// SIMATIC S7-200 project (STEP 7-Micro/WIN), CPU 222 REL 02.01

SYMBOL_TABLE 用户定义1
过程值              VD0
设定值              VD4
增益               VD8
采样时间             VD12
积分时间             VD16
微分时间             VD20
PID输出            VD24
积分前项             VD28
过程值前值            VD32
END_SYMBOL_TABLE

ORGANIZATION_BLOCK 主程序:OB1
TITLE=程序注释
BEGIN
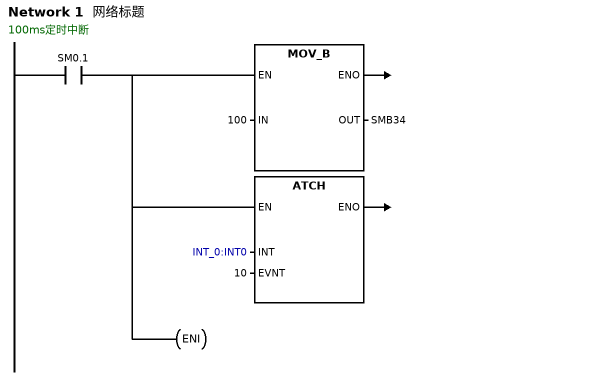
Network 1 // 网络标题
// 100ms定时中断
LD     SM0.1
MOVB   100, SMB34
ATCH   INT_0:INT0, 10
ENI
END_ORGANIZATION_BLOCK

SUBROUTINE_BLOCK PID调用:SBR0
TITLE=子程序注释
VAR_INPUT
过程值:REAL;	// LD0 
设定值:REAL;	// LD4 
增益:REAL;	// LD8 
采样时间:REAL;	// LD12 
积分时间:REAL;	// LD16 
微分时间:REAL;	// LD20 
END_VAR
VAR_IN_OUT
输出值:REAL;	// LD24 
积分前项:REAL;	// LD28 
过程值前值:REAL;	// LD32 
END_VAR
VAR
比例项:REAL;	// LD36 
积分项:REAL;	// LD40 
微分项:REAL;	// LD44 
END_VAR
BEGIN
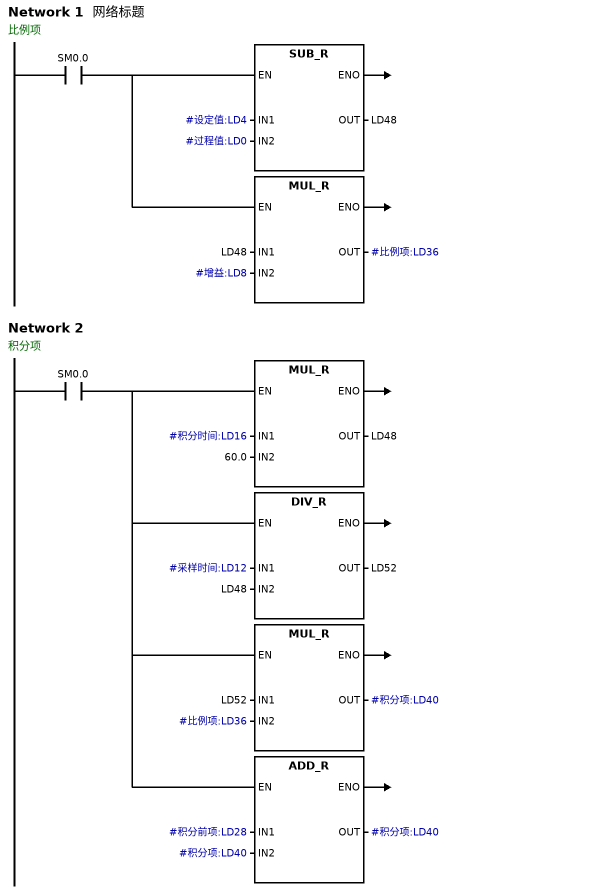
Network 1 // 网络标题
// 比例项
LD     SM0.0
MOVR   #设定值:LD4, LD48
-R     #过程值:LD0, LD48
MOVR   LD48, #比例项:LD36
*R     #增益:LD8, #比例项:LD36
Network 2
// 积分项
LD     SM0.0
MOVR   #积分时间:LD16, LD48
*R     60.0, LD48
MOVR   #采样时间:LD12, LD52
/R     LD48, LD52
MOVR   LD52, #积分项:LD40
*R     #比例项:LD36, #积分项:LD40
+R     #积分前项:LD28, #积分项:LD40
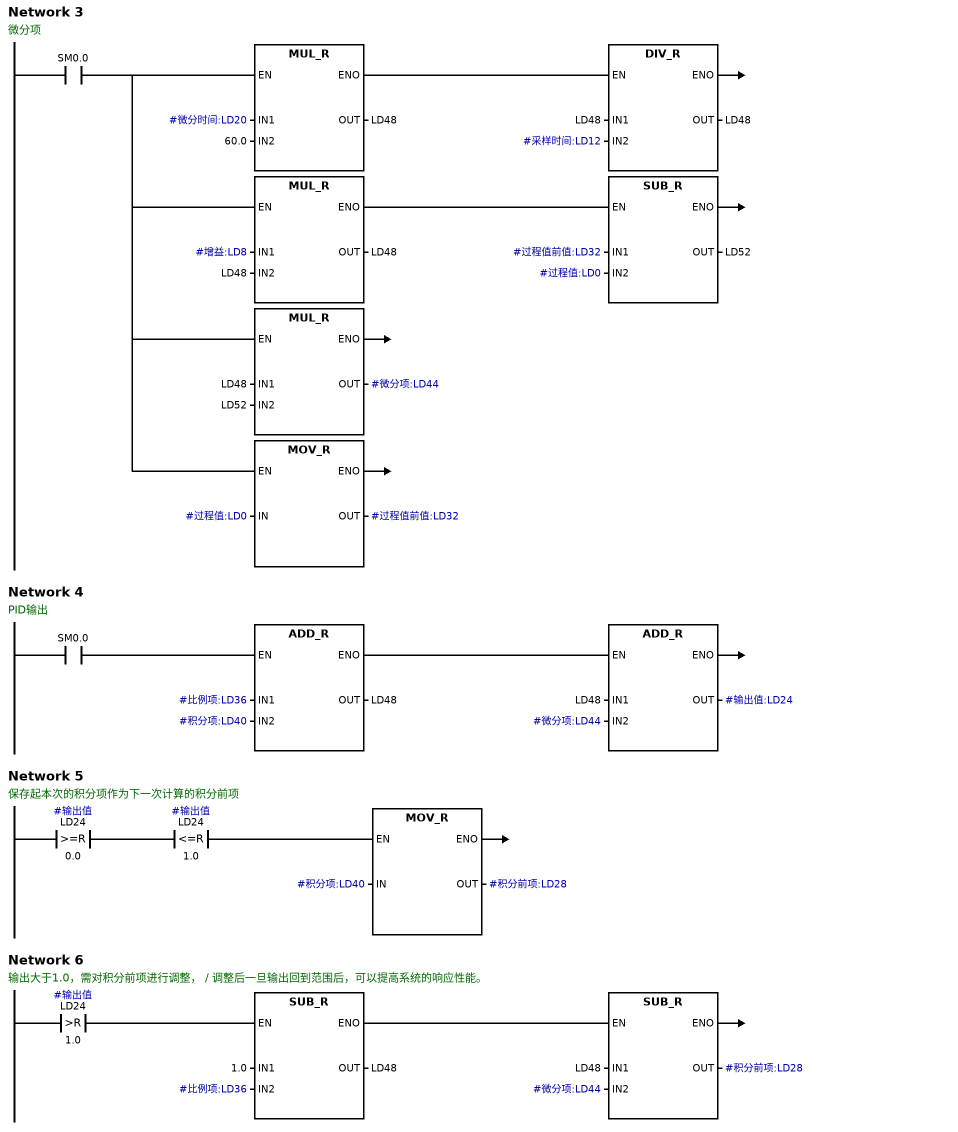
Network 3
// 微分项
LD     SM0.0
LPS
MOVR   #微分时间:LD20, LD48
AENO
*R     60.0, LD48
AENO
/R     #采样时间:LD12, LD48
LRD
*R     #增益:LD8, LD48
AENO
MOVR   #过程值前值:LD32, LD52
-R     #过程值:LD0, LD52
LRD
MOVR   LD48, #微分项:LD44
*R     LD52, #微分项:LD44
LPP
MOVR   #过程值:LD0, #过程值前值:LD32
Network 4
// PID输出
LD     SM0.0
MOVR   #比例项:LD36, LD48
AENO
+R     #积分项:LD40, LD48
AENO
MOVR   LD48, #输出值:LD24
+R     #微分项:LD44, #输出值:LD24
Network 5
// 保存起本次的积分项作为下一次计算的积分前项
LDR>=  #输出值:LD24, 0.0
AR<=   #输出值:LD24, 1.0
MOVR   #积分项:LD40, #积分前项:LD28
Network 6
// 输出大于1.0，需对积分前项进行调整，
// 调整后一旦输出回到范围后，可以提高系统的响应性能。
LDR>   #输出值:LD24, 1.0
MOVR   1.0, LD48
AENO
-R     #比例项:LD36, LD48
AENO
MOVR   LD48, #积分前项:LD28
-R     #微分项:LD44, #积分前项:LD28
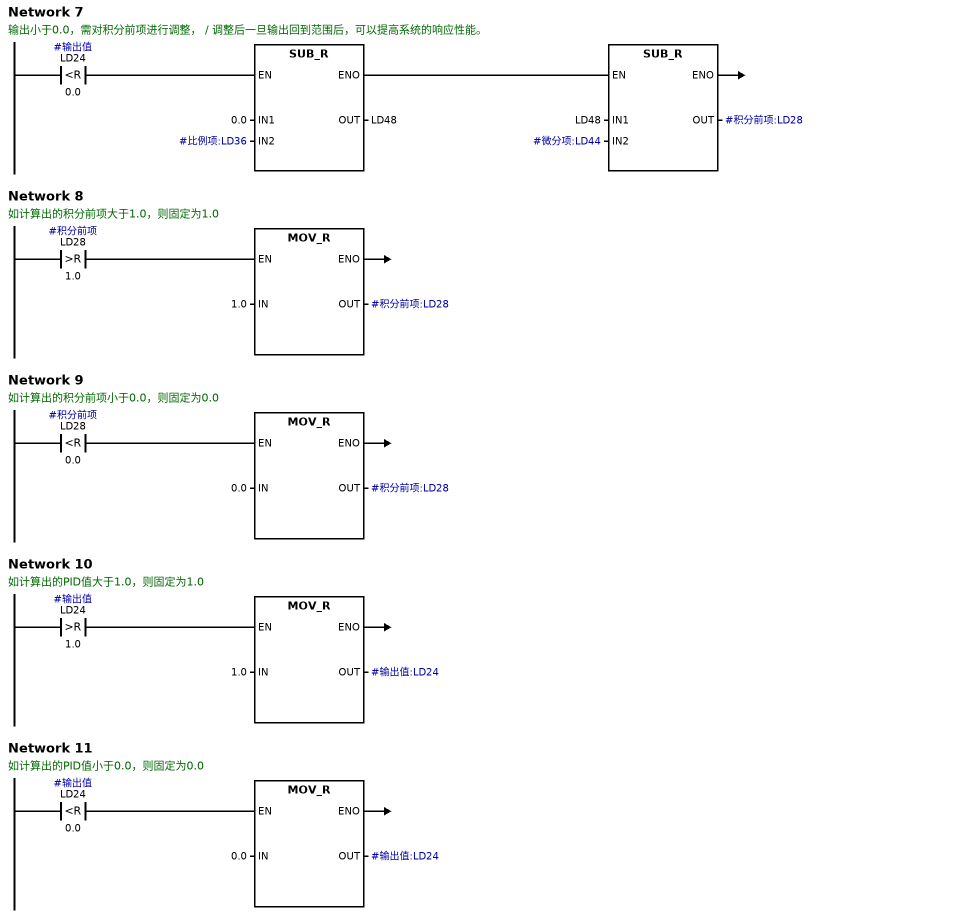
Network 7
// 输出小于0.0，需对积分前项进行调整，
// 调整后一旦输出回到范围后，可以提高系统的响应性能。
LDR<   #输出值:LD24, 0.0
MOVR   0.0, LD48
AENO
-R     #比例项:LD36, LD48
AENO
MOVR   LD48, #积分前项:LD28
-R     #微分项:LD44, #积分前项:LD28
Network 8
// 如计算出的积分前项大于1.0，则固定为1.0
LDR>   #积分前项:LD28, 1.0
MOVR   1.0, #积分前项:LD28
Network 9
// 如计算出的积分前项小于0.0，则固定为0.0
LDR<   #积分前项:LD28, 0.0
MOVR   0.0, #积分前项:LD28
Network 10
// 如计算出的PID值大于1.0，则固定为1.0
LDR>   #输出值:LD24, 1.0
MOVR   1.0, #输出值:LD24
Network 11
// 如计算出的PID值小于0.0，则固定为0.0
LDR<   #输出值:LD24, 0.0
MOVR   0.0, #输出值:LD24
END_SUBROUTINE_BLOCK

INTERRUPT_BLOCK INT_0:INT0
TITLE=中断程序注释
BEGIN
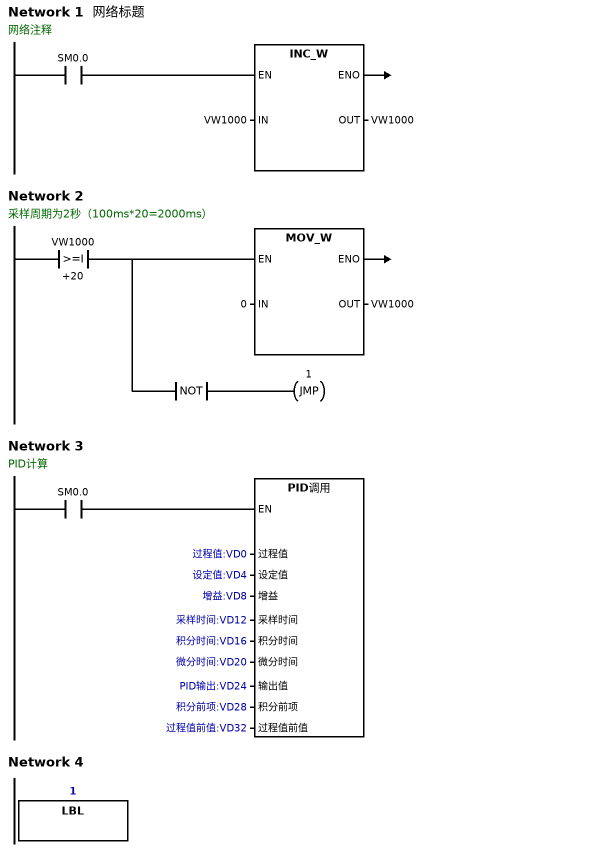
Network 1 // 网络标题
// 网络注释
LD     SM0.0
INCW   VW1000
Network 2
// 采样周期为2秒（100ms*20=2000ms）
LDW>=  VW1000, +20
MOVW   0, VW1000
NOT
JMP    1
Network 3
// PID计算
LD     SM0.0
CALL   PID调用:SBR0, 过程值:VD0, 设定值:VD4, 增益:VD8, 采样时间:VD12, 积分时间:VD16, 微分时间:VD20, PID输出:VD24, 积分前项:VD28, 过程值前值:VD32
Network 4
LBL    1
END_INTERRUPT_BLOCK
